// TIA Portal V17 export
// export: Created 2024-06-14T09:53:02.2081263Z, ExportSetting WithDefaults, DisplayName Totally Integrated Automation Portal, DisplayVersion V17, DisplayName TIA Portal Openness, DisplayVersion V17, DisplayName TIA Portal Version Control Interface, DisplayVersion V17, DisplayName Simotion SCOUT TIA, DisplayVersion 5.4.3.0, DisplayName SINAMICS Startdrive Advanced, DisplayVersion V17 SP1 Update 1, DisplayName SINAMICS Startdrive G110M, G120, G120C, G120D, G120P, G115D, DisplayVersion V17 SP1 Update 1, DisplayName SINAMICS Startdrive G130, G150, S120, S150, SINAMICS MV, S210, DisplayVersion V17 SP1 Update 1, DisplayName STEP 7 Professional, DisplayVersion V17, DisplayName STEP 7 Safety, DisplayVersion V17, DisplayName WinCC Professional, DisplayVersion V17
DATA_BLOCK "ALARM_DB_L2"   // DB505
{ S7_Optimized_Access := 'FALSE' }
VERSION : 0.1
// stored: AutoNumber false, DBAccessibleFromOPCUA true, IsOnlyStoredInLoadMemory false, IsWriteProtectedInAS false
   VAR
      COMMON_ALM1 : Word;
      COMMON_ALM2 : Word;
      S1_ALARM1 : Word;
      S1_ALARM2 : Word;
      S2_ALM1 : Word;
      S2_ALM2 : Word;
      S3_ALM1 : Word;
      S3_ALM2 : Word;
      S5_ALARM_STN1 : Word;
      S5_ALARM_STN2 : Word;
      S5_ALARM_STN3 : Word;
      S5_ALARM_STN4 : Word;
      S5_ALARM_STN5 : Word;
      S5_ALARM_STN6 : Word;
      S5_ALARM_STN7 : Word;
      S5_ALARM_STN8 : Word;
      S5_ALARM_STN9 : Word;
      S5_ALARM_STN10 : Word;
      S5_ALARM : Word;
   END_VAR
BEGIN
END_DATA_BLOCK
